// TIA Portal project "NastroTrasportatoreFB" (V16)

(* hardware
DEVICE "S7-1200 station_1"  S7-1200 Station
   slot 0: "Telaio di montaggio_0"  S7-1200 Rack  Rack  V1.0
   slot 1: "PLC_1"  CPU 1214C DC/DC/DC  6ES7 214-1AG40-0XB0  V4.1
*)

// ===== PLC "PLC_1"  CPU 1214C DC/DC/DC =====

VAR_GLOBAL   // PLC tag table "Tabella delle variabili standard"
   "START_1" AT %I0.0 : Bool;
   "S1_1" AT %I0.1 : Bool;
   "S2_1" AT %I0.2 : Bool;
   "S3_1" AT %I0.3 : Bool;
   "PRELIEVO_1" AT %M0.0 : Bool;
   "MOTOR_1" AT %Q0.0 : Bool;
   "START_2" AT %I0.4 : Bool;
   "S1_2" AT %I0.5 : Bool;
   "S2_2" AT %I0.6 : Bool;
   "S3_2" AT %I0.7 : Bool;
   "PRELIEVO_2" AT %M0.1 : Bool;
   "MOTOR_2" AT %Q0.1 : Bool;
END_VAR

VAR_GLOBAL CONSTANT   // PLC tag table "Tabella delle variabili standard"
   "TEMPO_TRASCORSO_T1_NastroTrasportatore1" : Time := T#5s;
   "TEMPO_TRASCORSO_T2_NastroTrasportatore2" : Time := T#10s;
END_VAR

DATA_BLOCK "NastroTrasportatore_DB_1"   // DB1
{ S7_Optimized_Access := 'TRUE' }
VERSION : 0.1
// stored: InstanceOfName NastroTrasportatore
"NastroTrasportatore"
BEGIN
END_DATA_BLOCK

DATA_BLOCK "NastroTrasportatore_DB_2"   // DB2
{ S7_Optimized_Access := 'TRUE' }
VERSION : 0.1
// stored: InstanceOfName NastroTrasportatore
"NastroTrasportatore"
BEGIN
END_DATA_BLOCK

FUNCTION_BLOCK "NastroTrasportatore"   // FB1, LAD
{ S7_Optimized_Access := 'TRUE' }
VERSION : 0.1
   VAR_INPUT
      START : Bool;
      S1 : Bool;
      S2 : Bool;
      S3 : Bool;
      TEMPO_TRASCORSO : Time;
   END_VAR
   VAR_OUTPUT
      MOTOR : Bool;
   END_VAR
   VAR_IN_OUT
      PRELIEVO : Bool;
   END_VAR
   VAR RETAIN
      HOME : Bool := true;
      MOVE_TO_S2 : Bool;
      POSITION_S2 : Bool;
      MOVE_TO_S3 : Bool;
      POSITION_TO_S3 : Bool;
   END_VAR
   VAR
      IEC_Timer_0_Instance : TON_TIME;
   END_VAR
BEGIN

REGION Network 1
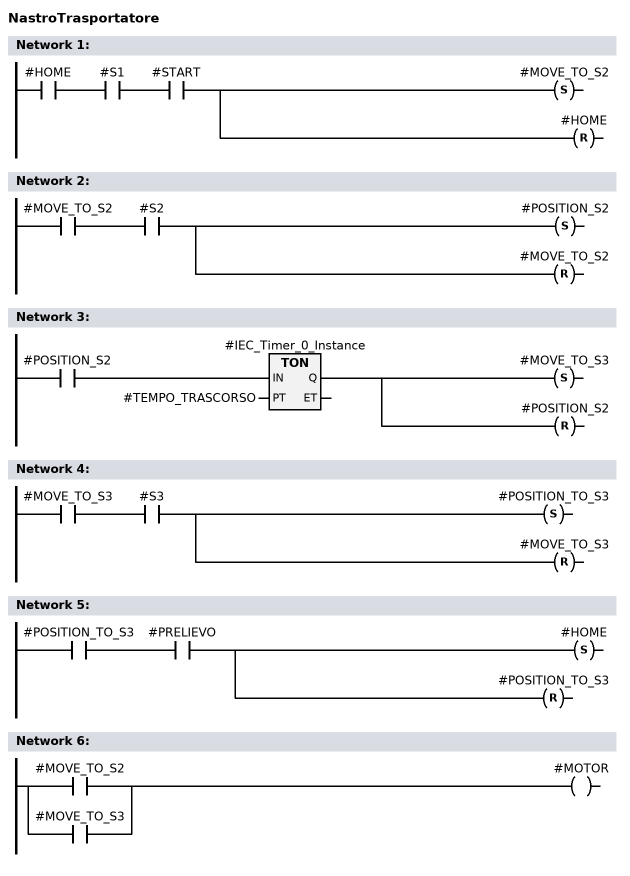
   RUNG wire#powerrail
      Contact( #HOME )
      Contact( #S1 )
      Contact( #START )
      wire#w1
      S_Coil( #MOVE_TO_S2 )
   END_RUNG
   RUNG wire#w1
      R_Coil( #HOME )
   END_RUNG
   // the same network as SCL:
   IF #HOME AND #S1 AND #START THEN
       #MOVE_TO_S2 := TRUE;
       #HOME := FALSE;
   END_IF;
END_REGION

REGION Network 2
   RUNG wire#powerrail
      Contact( #MOVE_TO_S2 )
      Contact( #S2 )
      wire#w1
      S_Coil( #POSITION_S2 )
   END_RUNG
   RUNG wire#w1
      R_Coil( #MOVE_TO_S2 )
   END_RUNG
   // the same network as SCL:
   IF #MOVE_TO_S2 AND #S2 THEN
       #POSITION_S2 := TRUE;
       #MOVE_TO_S2 := FALSE;
   END_IF;
END_REGION

REGION Network 3
   #IEC_Timer_0_Instance(IN := #POSITION_S2, PT := #TEMPO_TRASCORSO);   // TON
   IF #IEC_Timer_0_Instance.Q THEN
       #MOVE_TO_S3 := TRUE;
       #POSITION_S2 := FALSE;
   END_IF;
END_REGION

REGION Network 4
   RUNG wire#powerrail
      Contact( #MOVE_TO_S3 )
      Contact( #S3 )
      wire#w1
      S_Coil( #POSITION_TO_S3 )
   END_RUNG
   RUNG wire#w1
      R_Coil( #MOVE_TO_S3 )
   END_RUNG
   // the same network as SCL:
   IF #MOVE_TO_S3 AND #S3 THEN
       #POSITION_TO_S3 := TRUE;
       #MOVE_TO_S3 := FALSE;
   END_IF;
END_REGION

REGION Network 5
   RUNG wire#powerrail
      Contact( #POSITION_TO_S3 )
      Contact( #PRELIEVO )
      wire#w1
      S_Coil( #HOME )
   END_RUNG
   RUNG wire#w1
      R_Coil( #POSITION_TO_S3 )
   END_RUNG
   // the same network as SCL:
   IF #POSITION_TO_S3 AND #PRELIEVO THEN
       #HOME := TRUE;
       #POSITION_TO_S3 := FALSE;
   END_IF;
END_REGION

REGION Network 6
   RUNG wire#powerrail
      Contact( #MOVE_TO_S2 )
      wire#w1
      Coil( #MOTOR )
   END_RUNG
   RUNG wire#powerrail
      Contact( #MOVE_TO_S3 )
   END_RUNG wire#w1
   // the same network as SCL:
   #MOTOR := #MOVE_TO_S2 OR #MOVE_TO_S3;
END_REGION
END_FUNCTION_BLOCK

ORGANIZATION_BLOCK "Main"   // OB1, LAD, ProgramCycle
TITLE = "Main Program Sweep (Cycle)"
{ S7_Optimized_Access := 'TRUE' }
VERSION : 0.1
   VAR_INPUT
      Initial_Call : Bool;   // Initial call of this OB
      Remanence : Bool;   // =True, if remanent data are available
   END_VAR
BEGIN
END_ORGANIZATION_BLOCK

ORGANIZATION_BLOCK "Cyclic_Interrupt_50ms"   // OB30, LAD, CyclicInterrupt
{ S7_Optimized_Access := 'TRUE' }
VERSION : 0.1
   VAR_INPUT
      Initial_Call : Bool;   // Initial call of this OB
      Event_Count : Int;   // Events discarded
   END_VAR
BEGIN

REGION Network 1
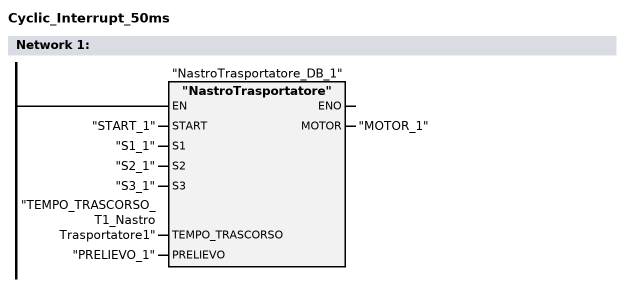
   RUNG wire#powerrail
      "NastroTrasportatore_DB_1"(START := "START_1", S1 := "S1_1", S2 := "S2_1", S3 := "S3_1", TEMPO_TRASCORSO := "TEMPO_TRASCORSO_T1_NastroTrasportatore1", PRELIEVO := "PRELIEVO_1", MOTOR => "MOTOR_1")
   END_RUNG
   // the same network as SCL:
   "NastroTrasportatore_DB_1"(START := "START_1",   // "NastroTrasportatore"
                           S1 := "S1_1",
                           S2 := "S2_1",
                           S3 := "S3_1",
                           TEMPO_TRASCORSO := "TEMPO_TRASCORSO_T1_NastroTrasportatore1",
                           PRELIEVO := "PRELIEVO_1",
                           MOTOR => "MOTOR_1");
END_REGION
END_ORGANIZATION_BLOCK

ORGANIZATION_BLOCK "Cyclic_Interrupt_100ms"   // OB31, LAD, CyclicInterrupt
{ S7_Optimized_Access := 'TRUE' }
VERSION : 0.1
   VAR_INPUT
      Initial_Call : Bool;   // Initial call of this OB
      Event_Count : Int;   // Events discarded
   END_VAR
BEGIN

REGION Network 1
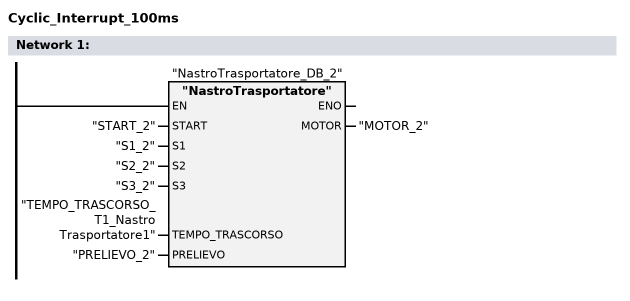
   RUNG wire#powerrail
      "NastroTrasportatore_DB_2"(START := "START_2", S1 := "S1_2", S2 := "S2_2", S3 := "S3_2", TEMPO_TRASCORSO := "TEMPO_TRASCORSO_T1_NastroTrasportatore1", PRELIEVO := "PRELIEVO_2", MOTOR => "MOTOR_2")
   END_RUNG
   // the same network as SCL:
   "NastroTrasportatore_DB_2"(START := "START_2",   // "NastroTrasportatore"
                           S1 := "S1_2",
                           S2 := "S2_2",
                           S3 := "S3_2",
                           TEMPO_TRASCORSO := "TEMPO_TRASCORSO_T1_NastroTrasportatore1",
                           PRELIEVO := "PRELIEVO_2",
                           MOTOR => "MOTOR_2");
END_REGION
END_ORGANIZATION_BLOCK

ORGANIZATION_BLOCK "Hardware_Interrupt_1"   // OB40, LAD, HWProcessInterrupt
{ S7_Optimized_Access := 'TRUE' }
VERSION : 0.1
   VAR_INPUT
      LADDR : Hw_Io;   // Hardware identifier
      USI : Word;   // User structure identifier
      IChannel : USInt;   // Interrupt channel number
      EventType : Byte;   // EventType
   END_VAR
BEGIN

REGION Network 1
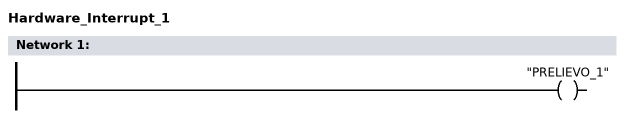
   RUNG wire#powerrail
      Coil( "PRELIEVO_1" )
   END_RUNG
   // the same network as SCL:
   "PRELIEVO_1" := TRUE;
END_REGION
END_ORGANIZATION_BLOCK

ORGANIZATION_BLOCK "Hardware_Interrupt_2"   // OB41, LAD, HWProcessInterrupt
{ S7_Optimized_Access := 'TRUE' }
VERSION : 0.1
   VAR_INPUT
      LADDR : Hw_Io;   // Hardware identifier
      USI : Word;   // User structure identifier
      IChannel : USInt;   // Interrupt channel number
      EventType : Byte;   // EventType
   END_VAR
BEGIN

REGION Network 1
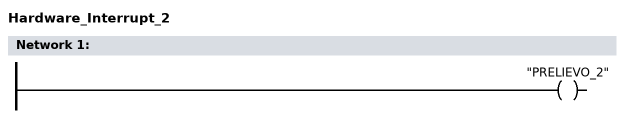
   RUNG wire#powerrail
      Coil( "PRELIEVO_2" )
   END_RUNG
   // the same network as SCL:
   "PRELIEVO_2" := TRUE;
END_REGION
END_ORGANIZATION_BLOCK